Universal Robots PolyScope program: all_seeing_run.urp

Program all_seeing_run (installation=default directory=/programs/usbdisk createdIn=5.12.4.1101661 lastSavedIn=5.12.4.1101661)
Robot Program (runOnlyOnce=true)
  Script file /programs/usbdisk/all_seeing.script
    | def draw_svg():
    |   draw_z = 0.074940
    |   # home
    |   movel(p[0.598550, -0.129200, 0.105150, 2.249000, -2.194000, 0.000000], a=0.8, v=0.25, r=0.0)
    |   # stroke 0 (form id 0): path
    |   movel(p[0.549770, -0.094886, 0.118080, 2.230000, -2.212000, 0.000000], a=0.8, v=0.25, r=0.0)
    |   movep(p[0.549770, -0.094886, draw_z, 2.230000, -2.212000, 0.000000], a=0.5, v=0.02, r=0.002472)
    |   movep(p[0.552918, -0.098699, draw_z, 2.230000, -2.212000, 0.000000], a=0.5, v=0.02, r=0.005327)
    |   movep(p[0.560362, -0.106321, draw_z, 2.230000, -2.212000, 0.000000], a=0.5, v=0.02, r=0.005323)
    |   movep(p[0.568940, -0.112625, draw_z, 2.230000, -2.212000, 0.000000], a=0.5, v=0.02, r=0.005331)
    |   movep(p[0.578444, -0.117461, draw_z, 2.230000, -2.212000, 0.000000], a=0.5, v=0.02, r=0.005313)
    |   movep(p[0.588577, -0.120662, draw_z, 2.230000, -2.212000, 0.000000], a=0.5, v=0.02, r=0.005295)
    |   movep(p[0.599059, -0.122174, draw_z, 2.230000, -2.212000, 0.000000], a=0.5, v=0.02, r=0.005300)
    |   movep(p[0.609657, -0.122002, draw_z, 2.230000, -2.212000, 0.000000], a=0.5, v=0.02, r=0.005321)
    |   movep(p[0.620137, -0.120149, draw_z, 2.230000, -2.212000, 0.000000], a=0.5, v=0.02, r=0.005363)
    |   movep(p[0.630264, -0.116618, draw_z, 2.230000, -2.212000, 0.000000], a=0.5, v=0.02, r=0.005393)
    |   movep(p[0.639744, -0.111473, draw_z, 2.230000, -2.212000, 0.000000], a=0.5, v=0.02, r=0.005395)
    |   movep(p[0.648293, -0.104890, draw_z, 2.230000, -2.212000, 0.000000], a=0.5, v=0.02, r=0.005402)
    |   movep(p[0.655702, -0.097027, draw_z, 2.230000, -2.212000, 0.000000], a=0.5, v=0.02, r=0.005013)
    |   movep(p[0.661963, -0.089197, draw_z, 2.230000, -2.212000, 0.000000], a=0.5, v=0.02, r=0.002914)
    |   movep(p[0.663479, -0.083570, draw_z, 2.230000, -2.212000, 0.000000], a=0.5, v=0.02, r=0.002880)
    |   movep(p[0.660349, -0.078735, draw_z, 2.230000, -2.212000, 0.000000], a=0.5, v=0.02, r=0.015000)
    |   movep(p[0.634236, -0.061822, draw_z, 2.230000, -2.212000, 0.000000], a=0.5, v=0.02, r=0.005353)
    |   movep(p[0.624719, -0.056920, draw_z, 2.230000, -2.212000, 0.000000], a=0.5, v=0.02, r=0.005252)
    |   movep(p[0.614613, -0.054053, draw_z, 2.230000, -2.212000, 0.000000], a=0.5, v=0.02, r=0.005219)
    |   movep(p[0.604208, -0.053213, draw_z, 2.230000, -2.212000, 0.000000], a=0.5, v=0.02, r=0.005233)
    |   movep(p[0.593807, -0.054391, draw_z, 2.230000, -2.212000, 0.000000], a=0.5, v=0.02, r=0.005293)
    |   movep(p[0.583715, -0.057586, draw_z, 2.230000, -2.212000, 0.000000], a=0.5, v=0.02, r=0.005415)
    |   movep(p[0.574221, -0.062798, draw_z, 2.230000, -2.212000, 0.000000], a=0.5, v=0.02, r=0.015000)
    |   movep(p[0.548188, -0.080559, draw_z, 2.230000, -2.212000, 0.000000], a=0.5, v=0.02, r=0.002917)
    |   movep(p[0.545080, -0.085496, draw_z, 2.230000, -2.212000, 0.000000], a=0.5, v=0.02, r=0.002893)
    |   movep(p[0.546622, -0.091073, draw_z, 2.230000, -2.212000, 0.000000], a=0.5, v=0.02, r=0.002472)
    |   movep(p[0.549770, -0.094886, draw_z, 2.230000, -2.212000, 0.000000], a=0.5, v=0.02, r=0.000000)
    |   movel(p[0.549770, -0.094886, 0.118080, 2.230000, -2.212000, 0.000000], a=0.8, v=0.25, r=0.0)
    |   # stroke 1 (form id 1): path
    |   movel(p[0.582103, -0.080497, 0.118080, 2.230000, -2.212000, 0.000000], a=0.8, v=0.25, r=0.0)
    |   movep(p[0.582103, -0.080497, draw_z, 2.230000, -2.212000, 0.000000], a=0.5, v=0.02, r=0.002676)
    |   movep(p[0.582985, -0.085776, draw_z, 2.230000, -2.212000, 0.000000], a=0.5, v=0.02, r=0.004413)
    |   movep(p[0.587962, -0.093066, draw_z, 2.230000, -2.212000, 0.000000], a=0.5, v=0.02, r=0.004409)
    |   movep(p[0.595323, -0.097921, draw_z, 2.230000, -2.212000, 0.000000], a=0.5, v=0.02, r=0.004573)
    |   movep(p[0.604314, -0.099600, draw_z, 2.230000, -2.212000, 0.000000], a=0.5, v=0.02, r=0.004523)
    |   movep(p[0.613156, -0.097692, draw_z, 2.230000, -2.212000, 0.000000], a=0.5, v=0.02, r=0.004543)
    |   movep(p[0.620644, -0.092545, draw_z, 2.230000, -2.212000, 0.000000], a=0.5, v=0.02, r=0.004548)
    |   movep(p[0.625638, -0.084943, draw_z, 2.230000, -2.212000, 0.000000], a=0.5, v=0.02, r=0.004534)
    |   movep(p[0.627378, -0.076043, draw_z, 2.230000, -2.212000, 0.000000], a=0.5, v=0.02, r=0.010650)
    |   movep(p[0.645913, -0.086536, draw_z, 2.230000, -2.212000, 0.000000], a=0.5, v=0.02, r=0.007381)
    |   movep(p[0.635553, -0.097052, draw_z, 2.230000, -2.212000, 0.000000], a=0.5, v=0.02, r=0.006337)
    |   movep(p[0.624668, -0.103544, draw_z, 2.230000, -2.212000, 0.000000], a=0.5, v=0.02, r=0.005256)
    |   movep(p[0.614674, -0.106800, draw_z, 2.230000, -2.212000, 0.000000], a=0.5, v=0.02, r=0.005209)
    |   movep(p[0.604326, -0.108000, draw_z, 2.230000, -2.212000, 0.000000], a=0.5, v=0.02, r=0.005193)
    |   movep(p[0.593976, -0.107137, draw_z, 2.230000, -2.212000, 0.000000], a=0.5, v=0.02, r=0.005209)
    |   movep(p[0.583979, -0.104206, draw_z, 2.230000, -2.212000, 0.000000], a=0.5, v=0.02, r=0.006261)
    |   movep(p[0.573063, -0.098069, draw_z, 2.230000, -2.212000, 0.000000], a=0.5, v=0.02, r=0.006268)
    |   movep(p[0.563946, -0.089464, draw_z, 2.230000, -2.212000, 0.000000], a=0.5, v=0.02, r=0.011196)
    |   movep(p[0.581222, -0.075217, draw_z, 2.230000, -2.212000, 0.000000], a=0.5, v=0.02, r=0.002676)
    |   movep(p[0.582103, -0.080497, draw_z, 2.230000, -2.212000, 0.000000], a=0.5, v=0.02, r=0.000000)
    |   movel(p[0.582103, -0.080497, 0.118080, 2.230000, -2.212000, 0.000000], a=0.8, v=0.25, r=0.0)
    |   # stroke 2 (form id 2): path
    |   movel(p[0.705292, -0.148351, 0.118080, 2.230000, -2.212000, 0.000000], a=0.8, v=0.25, r=0.0)
    |   movep(p[0.705292, -0.148351, draw_z, 2.230000, -2.212000, 0.000000], a=0.5, v=0.02, r=0.002594)
    |   movep(p[0.705042, -0.153533, draw_z, 2.230000, -2.212000, 0.000000], a=0.5, v=0.02, r=0.005098)
    |   movep(p[0.703530, -0.163616, draw_z, 2.230000, -2.212000, 0.000000], a=0.5, v=0.02, r=0.005030)
    |   movep(p[0.701057, -0.173368, draw_z, 2.230000, -2.212000, 0.000000], a=0.5, v=0.02, r=0.004980)
    |   movep(p[0.697673, -0.182737, draw_z, 2.230000, -2.212000, 0.000000], a=0.5, v=0.02, r=0.004945)
    |   movep(p[0.693429, -0.191669, draw_z, 2.230000, -2.212000, 0.000000], a=0.5, v=0.02, r=0.004920)
    |   movep(p[0.688378, -0.200114, draw_z, 2.230000, -2.212000, 0.000000], a=0.5, v=0.02, r=0.004905)
    |   movep(p[0.682569, -0.208018, draw_z, 2.230000, -2.212000, 0.000000], a=0.5, v=0.02, r=0.004897)
    |   movep(p[0.676054, -0.215330, draw_z, 2.230000, -2.212000, 0.000000], a=0.5, v=0.02, r=0.004895)
    |   movep(p[0.668884, -0.221997, draw_z, 2.230000, -2.212000, 0.000000], a=0.5, v=0.02, r=0.004901)
    |   movep(p[0.661111, -0.227967, draw_z, 2.230000, -2.212000, 0.000000], a=0.5, v=0.02, r=0.004914)
    |   movep(p[0.652784, -0.233188, draw_z, 2.230000, -2.212000, 0.000000], a=0.5, v=0.02, r=0.004936)
    |   movep(p[0.643956, -0.237608, draw_z, 2.230000, -2.212000, 0.000000], a=0.5, v=0.02, r=0.004970)
    |   movep(p[0.634678, -0.241174, draw_z, 2.230000, -2.212000, 0.000000], a=0.5, v=0.02, r=0.005018)
    |   movep(p[0.625000, -0.243835, draw_z, 2.230000, -2.212000, 0.000000], a=0.5, v=0.02, r=0.005085)
    |   movep(p[0.614973, -0.245537, draw_z, 2.230000, -2.212000, 0.000000], a=0.5, v=0.02, r=0.005173)
    |   movep(p[0.604650, -0.246230, draw_z, 2.230000, -2.212000, 0.000000], a=0.5, v=0.02, r=0.005166)
    |   movep(p[0.594324, -0.245873, draw_z, 2.230000, -2.212000, 0.000000], a=0.5, v=0.02, r=0.005064)
    |   movep(p[0.584291, -0.244497, draw_z, 2.230000, -2.212000, 0.000000], a=0.5, v=0.02, r=0.004985)
    |   movep(p[0.574601, -0.242151, draw_z, 2.230000, -2.212000, 0.000000], a=0.5, v=0.02, r=0.004925)
    |   movep(p[0.565307, -0.238887, draw_z, 2.230000, -2.212000, 0.000000], a=0.5, v=0.02, r=0.004883)
    |   movep(p[0.556460, -0.234755, draw_z, 2.230000, -2.212000, 0.000000], a=0.5, v=0.02, r=0.004853)
    |   movep(p[0.548110, -0.229805, draw_z, 2.230000, -2.212000, 0.000000], a=0.5, v=0.02, r=0.004836)
    |   movep(p[0.540309, -0.224088, draw_z, 2.230000, -2.212000, 0.000000], a=0.5, v=0.02, r=0.004828)
    |   movep(p[0.533110, -0.217655, draw_z, 2.230000, -2.212000, 0.000000], a=0.5, v=0.02, r=0.004829)
    |   movep(p[0.526562, -0.210556, draw_z, 2.230000, -2.212000, 0.000000], a=0.5, v=0.02, r=0.004839)
    |   movep(p[0.520717, -0.202841, draw_z, 2.230000, -2.212000, 0.000000], a=0.5, v=0.02, r=0.004859)
    |   movep(p[0.515627, -0.194562, draw_z, 2.230000, -2.212000, 0.000000], a=0.5, v=0.02, r=0.004891)
    |   movep(p[0.511343, -0.185768, draw_z, 2.230000, -2.212000, 0.000000], a=0.5, v=0.02, r=0.004936)
    |   movep(p[0.507916, -0.176510, draw_z, 2.230000, -2.212000, 0.000000], a=0.5, v=0.02, r=0.004997)
    |   movep(p[0.505398, -0.166839, draw_z, 2.230000, -2.212000, 0.000000], a=0.5, v=0.02, r=0.005077)
    |   movep(p[0.503840, -0.156805, draw_z, 2.230000, -2.212000, 0.000000], a=0.5, v=0.02, r=0.005180)
    |   movep(p[0.503293, -0.146459, draw_z, 2.230000, -2.212000, 0.000000], a=0.5, v=0.02, r=0.005059)
    |   movep(p[0.503770, -0.136353, draw_z, 2.230000, -2.212000, 0.000000], a=0.5, v=0.02, r=0.004973)
    |   movep(p[0.505213, -0.126512, draw_z, 2.230000, -2.212000, 0.000000], a=0.5, v=0.02, r=0.004908)
    |   movep(p[0.507574, -0.116984, draw_z, 2.230000, -2.212000, 0.000000], a=0.5, v=0.02, r=0.004860)
    |   movep(p[0.510804, -0.107817, draw_z, 2.230000, -2.212000, 0.000000], a=0.5, v=0.02, r=0.004825)
    |   movep(p[0.514852, -0.099058, draw_z, 2.230000, -2.212000, 0.000000], a=0.5, v=0.02, r=0.007958)
    |   movep(p[0.506019, -0.085819, draw_z, 2.230000, -2.212000, 0.000000], a=0.5, v=0.02, r=0.005219)
    |   movep(p[0.501002, -0.094971, draw_z, 2.230000, -2.212000, 0.000000], a=0.5, v=0.02, r=0.005246)
    |   movep(p[0.496796, -0.104584, draw_z, 2.230000, -2.212000, 0.000000], a=0.5, v=0.02, r=0.005285)
    |   movep(p[0.493447, -0.114609, draw_z, 2.230000, -2.212000, 0.000000], a=0.5, v=0.02, r=0.005337)
    |   movep(p[0.491004, -0.125001, draw_z, 2.230000, -2.212000, 0.000000], a=0.5, v=0.02, r=0.005407)
    |   movep(p[0.489514, -0.135710, draw_z, 2.230000, -2.212000, 0.000000], a=0.5, v=0.02, r=0.005496)
    |   movep(p[0.489024, -0.146692, draw_z, 2.230000, -2.212000, 0.000000], a=0.5, v=0.02, r=0.005261)
    |   movep(p[0.489520, -0.157202, draw_z, 2.230000, -2.212000, 0.000000], a=0.5, v=0.02, r=0.005166)
    |   movep(p[0.490934, -0.167436, draw_z, 2.230000, -2.212000, 0.000000], a=0.5, v=0.02, r=0.005089)
    |   movep(p[0.493223, -0.177354, draw_z, 2.230000, -2.212000, 0.000000], a=0.5, v=0.02, r=0.005029)
    |   movep(p[0.496347, -0.186914, draw_z, 2.230000, -2.212000, 0.000000], a=0.5, v=0.02, r=0.004982)
    |   movep(p[0.500265, -0.196076, draw_z, 2.230000, -2.212000, 0.000000], a=0.5, v=0.02, r=0.004947)
    |   movep(p[0.504935, -0.204799, draw_z, 2.230000, -2.212000, 0.000000], a=0.5, v=0.02, r=0.004923)
    |   movep(p[0.510316, -0.213044, draw_z, 2.230000, -2.212000, 0.000000], a=0.5, v=0.02, r=0.004907)
    |   movep(p[0.516368, -0.220769, draw_z, 2.230000, -2.212000, 0.000000], a=0.5, v=0.02, r=0.004898)
    |   movep(p[0.523048, -0.227934, draw_z, 2.230000, -2.212000, 0.000000], a=0.5, v=0.02, r=0.004897)
    |   movep(p[0.530316, -0.234499, draw_z, 2.230000, -2.212000, 0.000000], a=0.5, v=0.02, r=0.004903)
    |   movep(p[0.538131, -0.240422, draw_z, 2.230000, -2.212000, 0.000000], a=0.5, v=0.02, r=0.004917)
    |   movep(p[0.546451, -0.245665, draw_z, 2.230000, -2.212000, 0.000000], a=0.5, v=0.02, r=0.004940)
    |   movep(p[0.555235, -0.250185, draw_z, 2.230000, -2.212000, 0.000000], a=0.5, v=0.02, r=0.004973)
    |   movep(p[0.564443, -0.253943, draw_z, 2.230000, -2.212000, 0.000000], a=0.5, v=0.02, r=0.005017)
    |   movep(p[0.574033, -0.256898, draw_z, 2.230000, -2.212000, 0.000000], a=0.5, v=0.02, r=0.005076)
    |   movep(p[0.583963, -0.259010, draw_z, 2.230000, -2.212000, 0.000000], a=0.5, v=0.02, r=0.005152)
    |   movep(p[0.594194, -0.260237, draw_z, 2.230000, -2.212000, 0.000000], a=0.5, v=0.02, r=0.005247)
    |   movep(p[0.604683, -0.260541, draw_z, 2.230000, -2.212000, 0.000000], a=0.5, v=0.02, r=0.005253)
    |   movep(p[0.615170, -0.259896, draw_z, 2.230000, -2.212000, 0.000000], a=0.5, v=0.02, r=0.005171)
    |   movep(p[0.625394, -0.258336, draw_z, 2.230000, -2.212000, 0.000000], a=0.5, v=0.02, r=0.005107)
    |   movep(p[0.635314, -0.255901, draw_z, 2.230000, -2.212000, 0.000000], a=0.5, v=0.02, r=0.005059)
    |   movep(p[0.644889, -0.252635, draw_z, 2.230000, -2.212000, 0.000000], a=0.5, v=0.02, r=0.005023)
    |   movep(p[0.654079, -0.248577, draw_z, 2.230000, -2.212000, 0.000000], a=0.5, v=0.02, r=0.004997)
    |   movep(p[0.662842, -0.243771, draw_z, 2.230000, -2.212000, 0.000000], a=0.5, v=0.02, r=0.004980)
    |   movep(p[0.671138, -0.238259, draw_z, 2.230000, -2.212000, 0.000000], a=0.5, v=0.02, r=0.004970)
    |   movep(p[0.678925, -0.232081, draw_z, 2.230000, -2.212000, 0.000000], a=0.5, v=0.02, r=0.004966)
    |   movep(p[0.686162, -0.225281, draw_z, 2.230000, -2.212000, 0.000000], a=0.5, v=0.02, r=0.004967)
    |   movep(p[0.692809, -0.217899, draw_z, 2.230000, -2.212000, 0.000000], a=0.5, v=0.02, r=0.004973)
    |   movep(p[0.698825, -0.209977, draw_z, 2.230000, -2.212000, 0.000000], a=0.5, v=0.02, r=0.004986)
    |   movep(p[0.704168, -0.201558, draw_z, 2.230000, -2.212000, 0.000000], a=0.5, v=0.02, r=0.005005)
    |   movep(p[0.708797, -0.192683, draw_z, 2.230000, -2.212000, 0.000000], a=0.5, v=0.02, r=0.005032)
    |   movep(p[0.712673, -0.183395, draw_z, 2.230000, -2.212000, 0.000000], a=0.5, v=0.02, r=0.005070)
    |   movep(p[0.715753, -0.173734, draw_z, 2.230000, -2.212000, 0.000000], a=0.5, v=0.02, r=0.005120)
    |   movep(p[0.717997, -0.163743, draw_z, 2.230000, -2.212000, 0.000000], a=0.5, v=0.02, r=0.005185)
    |   movep(p[0.719363, -0.153464, draw_z, 2.230000, -2.212000, 0.000000], a=0.5, v=0.02, r=0.005268)
    |   movep(p[0.719812, -0.142938, draw_z, 2.230000, -2.212000, 0.000000], a=0.5, v=0.02, r=0.005489)
    |   movep(p[0.719271, -0.131972, draw_z, 2.230000, -2.212000, 0.000000], a=0.5, v=0.02, r=0.005386)
    |   movep(p[0.717732, -0.121312, draw_z, 2.230000, -2.212000, 0.000000], a=0.5, v=0.02, r=0.005304)
    |   movep(p[0.715241, -0.111001, draw_z, 2.230000, -2.212000, 0.000000], a=0.5, v=0.02, r=0.005240)
    |   movep(p[0.711847, -0.101085, draw_z, 2.230000, -2.212000, 0.000000], a=0.5, v=0.02, r=0.005192)
    |   movep(p[0.707597, -0.091610, draw_z, 2.230000, -2.212000, 0.000000], a=0.5, v=0.02, r=0.005157)
    |   movep(p[0.702539, -0.082622, draw_z, 2.230000, -2.212000, 0.000000], a=0.5, v=0.02, r=0.008061)
    |   movep(p[0.693767, -0.096148, draw_z, 2.230000, -2.212000, 0.000000], a=0.5, v=0.02, r=0.004774)
    |   movep(p[0.697856, -0.104775, draw_z, 2.230000, -2.212000, 0.000000], a=0.5, v=0.02, r=0.004817)
    |   movep(p[0.701127, -0.113837, draw_z, 2.230000, -2.212000, 0.000000], a=0.5, v=0.02, r=0.004876)
    |   movep(p[0.703531, -0.123287, draw_z, 2.230000, -2.212000, 0.000000], a=0.5, v=0.02, r=0.004953)
    |   movep(p[0.705019, -0.133080, draw_z, 2.230000, -2.212000, 0.000000], a=0.5, v=0.02, r=0.005052)
    |   movep(p[0.705542, -0.143170, draw_z, 2.230000, -2.212000, 0.000000], a=0.5, v=0.02, r=0.002594)
    |   movep(p[0.705292, -0.148351, draw_z, 2.230000, -2.212000, 0.000000], a=0.5, v=0.02, r=0.000000)
    |   movel(p[0.705292, -0.148351, 0.118080, 2.230000, -2.212000, 0.000000], a=0.8, v=0.25, r=0.0)
    |   # stroke 3 (form id 3): path
    |   movel(p[0.528845, -0.068234, 0.118080, 2.230000, -2.212000, 0.000000], a=0.8, v=0.25, r=0.0)
    |   movep(p[0.528845, -0.068234, draw_z, 2.230000, -2.212000, 0.000000], a=0.5, v=0.02, r=0.003606)
    |   movep(p[0.532847, -0.074234, draw_z, 2.230000, -2.212000, 0.000000], a=0.5, v=0.02, r=0.004889)
    |   movep(p[0.540014, -0.067581, draw_z, 2.230000, -2.212000, 0.000000], a=0.5, v=0.02, r=0.004895)
    |   movep(p[0.547783, -0.061623, draw_z, 2.230000, -2.212000, 0.000000], a=0.5, v=0.02, r=0.004908)
    |   movep(p[0.556102, -0.056413, draw_z, 2.230000, -2.212000, 0.000000], a=0.5, v=0.02, r=0.004930)
    |   movep(p[0.564922, -0.052003, draw_z, 2.230000, -2.212000, 0.000000], a=0.5, v=0.02, r=0.004964)
    |   movep(p[0.574191, -0.048445, draw_z, 2.230000, -2.212000, 0.000000], a=0.5, v=0.02, r=0.005013)
    |   movep(p[0.583858, -0.045790, draw_z, 2.230000, -2.212000, 0.000000], a=0.5, v=0.02, r=0.005079)
    |   movep(p[0.593873, -0.044091, draw_z, 2.230000, -2.212000, 0.000000], a=0.5, v=0.02, r=0.005167)
    |   movep(p[0.604185, -0.043399, draw_z, 2.230000, -2.212000, 0.000000], a=0.5, v=0.02, r=0.005160)
    |   movep(p[0.614499, -0.043755, draw_z, 2.230000, -2.212000, 0.000000], a=0.5, v=0.02, r=0.005058)
    |   movep(p[0.624521, -0.045128, draw_z, 2.230000, -2.212000, 0.000000], a=0.5, v=0.02, r=0.004979)
    |   movep(p[0.634200, -0.047468, draw_z, 2.230000, -2.212000, 0.000000], a=0.5, v=0.02, r=0.004920)
    |   movep(p[0.643485, -0.050725, draw_z, 2.230000, -2.212000, 0.000000], a=0.5, v=0.02, r=0.004877)
    |   movep(p[0.652324, -0.054848, draw_z, 2.230000, -2.212000, 0.000000], a=0.5, v=0.02, r=0.004848)
    |   movep(p[0.660667, -0.059787, draw_z, 2.230000, -2.212000, 0.000000], a=0.5, v=0.02, r=0.004830)
    |   movep(p[0.668462, -0.065491, draw_z, 2.230000, -2.212000, 0.000000], a=0.5, v=0.02, r=0.004822)
    |   movep(p[0.675659, -0.071911, draw_z, 2.230000, -2.212000, 0.000000], a=0.5, v=0.02, r=0.007305)
    |   movep(p[0.683608, -0.059651, draw_z, 2.230000, -2.212000, 0.000000], a=0.5, v=0.02, r=0.004732)
    |   movep(p[0.676431, -0.053483, draw_z, 2.230000, -2.212000, 0.000000], a=0.5, v=0.02, r=0.004739)
    |   movep(p[0.668756, -0.047921, draw_z, 2.230000, -2.212000, 0.000000], a=0.5, v=0.02, r=0.004754)
    |   movep(p[0.660618, -0.043003, draw_z, 2.230000, -2.212000, 0.000000], a=0.5, v=0.02, r=0.004777)
    |   movep(p[0.652055, -0.038767, draw_z, 2.230000, -2.212000, 0.000000], a=0.5, v=0.02, r=0.004809)
    |   movep(p[0.643104, -0.035248, draw_z, 2.230000, -2.212000, 0.000000], a=0.5, v=0.02, r=0.004852)
    |   movep(p[0.633802, -0.032483, draw_z, 2.230000, -2.212000, 0.000000], a=0.5, v=0.02, r=0.004909)
    |   movep(p[0.624184, -0.030511, draw_z, 2.230000, -2.212000, 0.000000], a=0.5, v=0.02, r=0.004981)
    |   movep(p[0.614289, -0.029367, draw_z, 2.230000, -2.212000, 0.000000], a=0.5, v=0.02, r=0.005070)
    |   movep(p[0.604152, -0.029089, draw_z, 2.230000, -2.212000, 0.000000], a=0.5, v=0.02, r=0.005076)
    |   movep(p[0.594018, -0.029697, draw_z, 2.230000, -2.212000, 0.000000], a=0.5, v=0.02, r=0.004999)
    |   movep(p[0.584128, -0.031163, draw_z, 2.230000, -2.212000, 0.000000], a=0.5, v=0.02, r=0.004938)
    |   movep(p[0.574521, -0.033448, draw_z, 2.230000, -2.212000, 0.000000], a=0.5, v=0.02, r=0.004891)
    |   movep(p[0.565231, -0.036514, draw_z, 2.230000, -2.212000, 0.000000], a=0.5, v=0.02, r=0.004856)
    |   movep(p[0.556297, -0.040324, draw_z, 2.230000, -2.212000, 0.000000], a=0.5, v=0.02, r=0.004831)
    |   movep(p[0.547755, -0.044839, draw_z, 2.230000, -2.212000, 0.000000], a=0.5, v=0.02, r=0.004814)
    |   movep(p[0.539640, -0.050021, draw_z, 2.230000, -2.212000, 0.000000], a=0.5, v=0.02, r=0.004803)
    |   movep(p[0.531991, -0.055832, draw_z, 2.230000, -2.212000, 0.000000], a=0.5, v=0.02, r=0.004798)
    |   movep(p[0.524842, -0.062234, draw_z, 2.230000, -2.212000, 0.000000], a=0.5, v=0.02, r=0.003606)
    |   movep(p[0.528845, -0.068234, draw_z, 2.230000, -2.212000, 0.000000], a=0.5, v=0.02, r=0.000000)
    |   movel(p[0.528845, -0.068234, 0.118080, 2.230000, -2.212000, 0.000000], a=0.8, v=0.25, r=0.0)
    |   # stroke 4 (form id 4): path
    |   movel(p[0.604037, 0.021141, 0.118080, 2.230000, -2.212000, 0.000000], a=0.8, v=0.25, r=0.0)
    |   movep(p[0.604037, 0.021141, draw_z, 2.230000, -2.212000, 0.000000], a=0.5, v=0.02, r=0.015000)
    |   movep(p[0.749793, 0.023511, draw_z, 2.230000, -2.212000, 0.000000], a=0.5, v=0.02, r=0.003640)
    |   movep(p[0.756085, 0.019850, draw_z, 2.230000, -2.212000, 0.000000], a=0.5, v=0.02, r=0.003672)
    |   movep(p[0.755775, 0.012513, draw_z, 2.230000, -2.212000, 0.000000], a=0.5, v=0.02, r=0.015000)
    |   movep(p[0.610527, -0.211472, draw_z, 2.230000, -2.212000, 0.000000], a=0.5, v=0.02, r=0.003405)
    |   movep(p[0.604578, -0.214785, draw_z, 2.230000, -2.212000, 0.000000], a=0.5, v=0.02, r=0.003365)
    |   movep(p[0.598614, -0.211666, draw_z, 2.230000, -2.212000, 0.000000], a=0.5, v=0.02, r=0.015000)
    |   movep(p[0.452350, 0.007578, draw_z, 2.230000, -2.212000, 0.000000], a=0.5, v=0.02, r=0.003667)
    |   movep(p[0.452007, 0.014904, draw_z, 2.230000, -2.212000, 0.000000], a=0.5, v=0.02, r=0.003685)
    |   movep(p[0.458281, 0.018770, draw_z, 2.230000, -2.212000, 0.000000], a=0.5, v=0.02, r=0.015000)
    |   movep(p[0.604037, 0.021141, draw_z, 2.230000, -2.212000, 0.000000], a=0.5, v=0.02, r=0.000000)
    |   movel(p[0.604037, 0.021141, 0.118080, 2.230000, -2.212000, 0.000000], a=0.8, v=0.25, r=0.0)
    |   # stroke 5 (form id 5): path
    |   movel(p[0.604070, 0.006830, 0.118080, 2.230000, -2.212000, 0.000000], a=0.8, v=0.25, r=0.0)
    |   movep(p[0.604070, 0.006830, draw_z, 2.230000, -2.212000, 0.000000], a=0.5, v=0.02, r=0.015000)
    |   movep(p[0.471567, 0.004674, draw_z, 2.230000, -2.212000, 0.000000], a=0.5, v=0.02, r=0.015000)
    |   movep(p[0.604532, -0.194635, draw_z, 2.230000, -2.212000, 0.000000], a=0.5, v=0.02, r=0.015000)
    |   movep(p[0.736573, 0.008985, draw_z, 2.230000, -2.212000, 0.000000], a=0.5, v=0.02, r=0.015000)
    |   movep(p[0.604070, 0.006830, draw_z, 2.230000, -2.212000, 0.000000], a=0.5, v=0.02, r=0.000000)
    |   movel(p[0.604070, 0.006830, 0.118080, 2.230000, -2.212000, 0.000000], a=0.8, v=0.25, r=0.0)
    |   # park
    |   movel(p[0.598550, -0.129200, 0.105150, 2.249000, -2.194000, 0.000000], a=0.8, v=0.25, r=0.0)
    | end
    | draw_svg()
